Staubli VAL3: RobotStatus.dtx

public JointSpace jointSpace
  [0]
    jointRx JointPos
    num JointVel[6]
    num JointAccel[6]
    num JointForce[6]
public CartesianSpace cartesianSpace
  [0]
    pointRx CartesianPos
    num CartesianVel[6]
    num CartesianAccel[6]
    num CartesianForce[6]
    num CarteResVel
    num CarteResAccel
    num CarteResForce
